FUNCTION_BLOCK CounterBasic (* Basic Function Block Type *)
  (* Standard: 61499-2 *)
  (* Version 0.0, 7/6/2026, Schneider Electric, Template *)
  PACKAGE SE.Nereda;
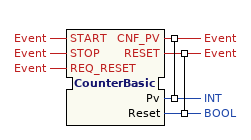
  EVENT_INPUT
    START; (* Normal Execution Request *)
    STOP;
    REQ_RESET;
  END_EVENT
  EVENT_OUTPUT
    CNF_PV WITH Pv; (* Execution Confirmation *)
    RESET WITH Reset;
  END_EVENT
  VAR_OUTPUT
    Pv : INT; (* Output event qualifier *)
    Reset : BOOL;
  END_VAR
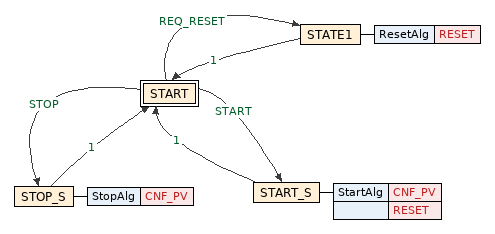
  EC_STATES
    START; (* Initial State *)
    START_S : StartAlg -> CNF_PV, -> RESET;
    STOP_S : StopAlg -> CNF_PV;
    STATE1 : ResetAlg -> RESET;
  END_STATES
  EC_TRANSITIONS
    START TO START_S := START;
    START_S TO START := 1;
    START TO STOP_S := STOP;
    STOP_S TO START := 1;
    START TO STATE1 := REQ_RESET;
    STATE1 TO START := 1;
  END_TRANSITIONS
  ALGORITHM StartAlg IN ST:
;
Pv := 1;
Reset := FALSE;
  END_ALGORITHM
  ALGORITHM StopAlg IN ST:
;
Pv := 0;
  END_ALGORITHM
  ALGORITHM ResetAlg IN ST:
;
Reset := TRUE;
  END_ALGORITHM
END_FUNCTION_BLOCK
